// TIA Portal project "Stat Remp 2essay" (V15)

(* hardware
DEVICE "HMI_1"  TP1200 Comfort
   slot 0: "HMI_1"  TP1200 Comfort  6AV2 124-0MC01-0AX0  15.0.0.0
   slot 1: "HMI_RT_1"  TP1200 Comfort  6AV2 124-0MC01-0AX0  15.0.0.0
   slot 5: "HMI_1.IE_CP_1"  PROFINET Interface  15.0.0.0
      slot 1: "Interface PROFINET_1"  PROFINET Interface
         slot 1: "Port_1"  Port
         slot 2: "Port_2"  Port
   slot 7: "HMI_1.MPI/DP_CP_1"  MPI/DP Interface  15.0.0.0
DEVICE "Station S7-1200_1"  S7-1200 Station
   slot 0: "Châssis_0"  S7-1200 Rack  Rack  V1.0
   slot 1: "PLC_1"  CPU 1214C DC/DC/DC  6ES7 214-1AG40-0XB0  V4.2
*)

// ===== PLC "PLC_1"  CPU 1214C DC/DC/DC =====

VAR_GLOBAL   // PLC tag table "Table de variables standard"
   "System_Byte" AT %MB1 : Byte;
   "FirstScan" AT %M1.0 : Bool;
   "DiagStatusUpdate" AT %M1.1 : Bool;
   "AlwaysTRUE" AT %M1.2 : Bool;
   "AlwaysFALSE" AT %M1.3 : Bool;
   "Clock_Byte" AT %MB0 : Byte;
   "Clock_10Hz" AT %M0.0 : Bool;
   "Clock_5Hz" AT %M0.1 : Bool;
   "Clock_2.5Hz" AT %M0.2 : Bool;
   "Clock_2Hz" AT %M0.3 : Bool;
   "Clock_1.25Hz" AT %M0.4 : Bool;
   "Clock_1Hz" AT %M0.5 : Bool;
   "Clock_0.625Hz" AT %M0.6 : Bool;
   "Clock_0.5Hz" AT %M0.7 : Bool;
   "X1" AT %M2.0 : Bool;
   "V1" AT %Q0.0 : Bool;
   "X2" AT %M2.1 : Bool;
   "V3" AT %Q0.1 : Bool;
   "X3" AT %M2.2 : Bool;
   "V2" AT %Q0.2 : Bool;
   "MM" AT %Q0.3 : Bool;
   "X4" AT %M2.3 : Bool;
   "X5" AT %M2.4 : Bool;
   "MP" AT %Q0.4 : Bool;
   "X6" AT %M2.5 : Bool;
   "V6" AT %Q0.5 : Bool;
   "X7" AT %M2.6 : Bool;
   "MDR" AT %Q0.6 : Bool;
   "X8" AT %M2.7 : Bool;
   "DC" AT %Q0.7 : Bool;
   "X9" AT %M3.0 : Bool;
   "MG" AT %Q1.0 : Bool;
   "M-PT100" AT %MW4 : Int;
   "NICH" AT %MD6 : Real;
   "TMP" AT %MW10 : Int;
   "NIVEAU" AT %MW12 : Int;
   "NIV" AT %MD14 : Real;
   "M-NIVEAU" AT %MW18 : Int;
   "X0" AT %M3.1 : Bool;
   "forçage" AT %M3.2 : Bool;
   "L50" AT %M3.3 : Bool;
   "L400" AT %M3.4 : Bool;
   "L900" AT %M3.5 : Bool;
   "MA" AT %M3.6 : Bool;
   "MIN1" AT %M3.7 : Bool;
   "MAX1" AT %M20.0 : Bool;
   "FC-CHARG" AT %M20.1 : Bool;
   "MAXC" AT %M20.2 : Bool;
   "FC-DECH" AT %M20.3 : Bool;
   "VASC" AT %Q1.1 : Bool;
   "VADN" AT %Q1.2 : Bool;
   "THR-P" AT %M20.4 : Bool;
   "VAP" AT %Q1.3 : Bool;
   "ALARME" AT %M56.0 : Bool;
   "Acquitt-Btn" AT %M20.5 : Bool;
   "Acquittement" AT %M58.0 : Bool;
   "Res-Alr" AT %M20.6 : Bool;
   "Stop" AT %M20.7 : Bool;
   "Mot-Alarme" AT %MW56 : Int;
   "Mot-Acquittement" AT %MW58 : Int;
END_VAR

// folder: System blocks/Program resources

DATA_BLOCK "T1"   // DB1
{ S7_Optimized_Access := 'TRUE' }
AUTHOR : Simatic
FAMILY : IEC
NAME : IEC_TMR
VERSION : 1.0
// stored: InstanceOfName IEC_TIMER
"IEC_TIMER"
BEGIN
END_DATA_BLOCK

DATA_BLOCK "T2"   // DB2
{ S7_Optimized_Access := 'TRUE' }
AUTHOR : Simatic
FAMILY : IEC
NAME : IEC_TMR
VERSION : 1.0
// stored: InstanceOfName IEC_TIMER
"IEC_TIMER"
BEGIN
END_DATA_BLOCK

DATA_BLOCK "T3"   // DB3
{ S7_Optimized_Access := 'TRUE' }
AUTHOR : Simatic
FAMILY : IEC
NAME : IEC_TMR
VERSION : 1.0
// stored: InstanceOfName IEC_TIMER
"IEC_TIMER"
BEGIN
END_DATA_BLOCK

// folder: (top level)

FUNCTION "Actions" : Void   // FC1, LAD
{ S7_Optimized_Access := 'TRUE' }
VERSION : 0.1
   VAR_TEMP   // added for the SCL form of the ladder/FBD networks
      _w1 : Bool;
   END_VAR
BEGIN

REGION Network 1
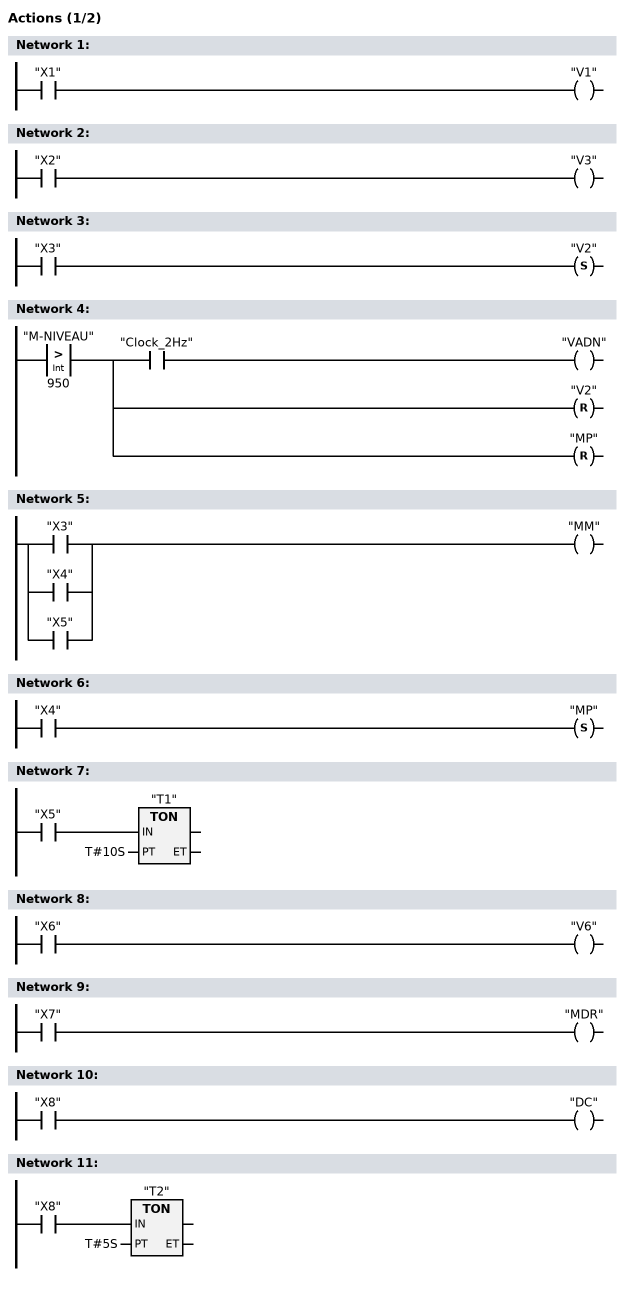
   RUNG wire#powerrail
      Contact( "X1" )
      Coil( "V1" )
   END_RUNG
   // the same network as SCL:
   "V1" := "X1";
END_REGION

REGION Network 2
   RUNG wire#powerrail
      Contact( "X2" )
      Coil( "V3" )
   END_RUNG
   // the same network as SCL:
   "V3" := "X2";
END_REGION

REGION Network 3
   RUNG wire#powerrail
      Contact( "X3" )
      S_Coil( "V2" )
   END_RUNG
   // the same network as SCL:
   IF "X3" THEN "V2" := TRUE; END_IF;
END_REGION

REGION Network 4
   RUNG wire#powerrail
      { S7_Templates := "SrcType := Int" } GT_Contact(in1 := "M-NIVEAU", in2 := 950)
      wire#w1
      Contact( "Clock_2Hz" )
      Coil( "VADN" )
   END_RUNG
   RUNG wire#w1
      R_Coil( "V2" )
   END_RUNG
   RUNG wire#w1
      R_Coil( "MP" )
   END_RUNG
   // the same network as SCL:
   #_w1 := "M-NIVEAU" > 950;
   "VADN" := #_w1 AND "Clock_2Hz";
   IF #_w1 THEN
       "V2" := FALSE;
       "MP" := FALSE;
   END_IF;
END_REGION

REGION Network 5
   RUNG wire#powerrail
      Contact( "X3" )
      wire#w1
      Coil( "MM" )
   END_RUNG
   RUNG wire#powerrail
      Contact( "X4" )
   END_RUNG wire#w1
   RUNG wire#powerrail
      Contact( "X5" )
   END_RUNG wire#w1
   // the same network as SCL:
   "MM" := "X3" OR "X4" OR "X5";
END_REGION

REGION Network 6
   RUNG wire#powerrail
      Contact( "X4" )
      S_Coil( "MP" )
   END_RUNG
   // the same network as SCL:
   IF "X4" THEN "MP" := TRUE; END_IF;
END_REGION

REGION Network 7
   "T1".TON(IN := "X5", PT := T#10S);
END_REGION

REGION Network 8
   RUNG wire#powerrail
      Contact( "X6" )
      Coil( "V6" )
   END_RUNG
   // the same network as SCL:
   "V6" := "X6";
END_REGION

REGION Network 9
   RUNG wire#powerrail
      Contact( "X7" )
      Coil( "MDR" )
   END_RUNG
   // the same network as SCL:
   "MDR" := "X7";
END_REGION

REGION Network 10
   RUNG wire#powerrail
      Contact( "X8" )
      Coil( "DC" )
   END_RUNG
   // the same network as SCL:
   "DC" := "X8";
END_REGION

REGION Network 11
   "T2".TON(IN := "X8", PT := T#5S);
END_REGION

REGION Network 12
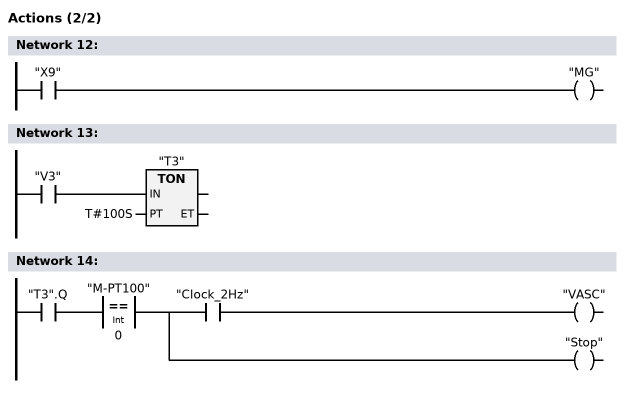
   RUNG wire#powerrail
      Contact( "X9" )
      Coil( "MG" )
   END_RUNG
   // the same network as SCL:
   "MG" := "X9";
END_REGION

REGION Network 13
   "T3".TON(IN := "V3", PT := T#100S);
END_REGION

REGION Network 14
   RUNG wire#powerrail
      Contact( "T3".Q )
      { S7_Templates := "SrcType := Int" } EQ_Contact(in1 := "M-PT100", in2 := 0)
      wire#w1
      Contact( "Clock_2Hz" )
      Coil( "VASC" )
   END_RUNG
   RUNG wire#w1
      Coil( "Stop" )
   END_RUNG
   // the same network as SCL:
   #_w1 := "T3".Q AND ("M-PT100" = 0);
   "VASC" := #_w1 AND "Clock_2Hz";
   "Stop" := #_w1;
END_REGION
END_FUNCTION

FUNCTION "Etapes" : Void   // FC2, LAD
{ S7_Optimized_Access := 'TRUE' }
VERSION : 0.1
BEGIN

REGION Network 1
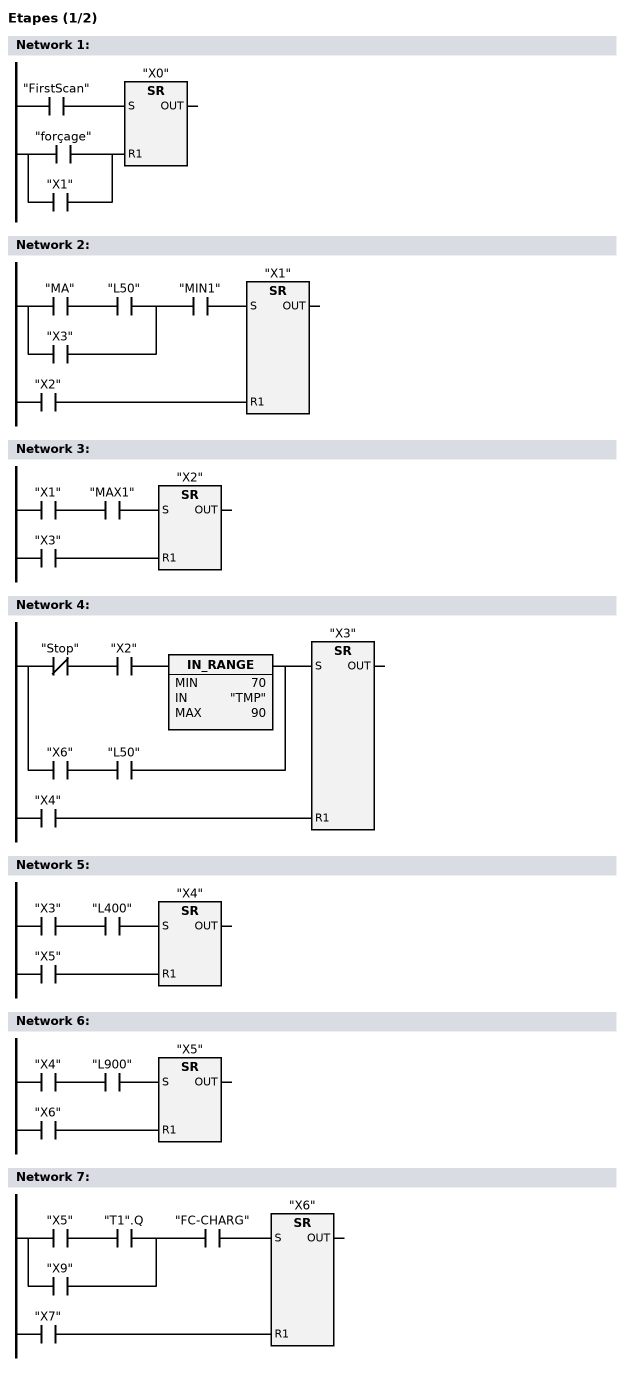
   RUNG wire#powerrail
      Contact( "FirstScan" )
      S_SR(operand := "X0", r1 := wire#w1)
   END_RUNG
   RUNG wire#powerrail
      Contact( "forçage" )
   END_RUNG wire#w1
   RUNG wire#powerrail
      Contact( "X1" )
   END_RUNG wire#w1
   // the same network as SCL:
   IF "FirstScan" THEN
       "X0" := TRUE;   // SR flip-flop
   END_IF;
   IF "forçage" OR "X1" THEN "X0" := FALSE; END_IF;
END_REGION

REGION Network 2
   RUNG wire#powerrail
      Contact( "MA" )
      Contact( "L50" )
      wire#w1
      Contact( "MIN1" )
      S_SR(operand := "X1", r1 := wire#w2)
   END_RUNG
   RUNG wire#powerrail
      Contact( "X3" )
   END_RUNG wire#w1
   RUNG wire#powerrail
      Contact( "X2" )
   END_RUNG wire#w2
   // the same network as SCL:
   IF (("MA" AND "L50") OR "X3") AND "MIN1" THEN
       "X1" := TRUE;   // SR flip-flop
   END_IF;
   IF "X2" THEN "X1" := FALSE; END_IF;
END_REGION

REGION Network 3
   RUNG wire#powerrail
      Contact( "X1" )
      Contact( "MAX1" )
      S_SR(operand := "X2", r1 := wire#w1)
   END_RUNG
   RUNG wire#powerrail
      Contact( "X3" )
   END_RUNG wire#w1
   // the same network as SCL:
   IF "X1" AND "MAX1" THEN
       "X2" := TRUE;   // SR flip-flop
   END_IF;
   IF "X3" THEN "X2" := FALSE; END_IF;
END_REGION

REGION Network 4
   RUNG wire#powerrail
      I_Contact( "Stop" )
      Contact( "X2" )
      { S7_Templates := "SrcType := Int" } InRange(min := 70, in := "TMP", max := 90)
      wire#w1
      S_SR(operand := "X3", r1 := wire#w2)
   END_RUNG
   RUNG wire#powerrail
      Contact( "X6" )
      Contact( "L50" )
   END_RUNG wire#w1
   RUNG wire#powerrail
      Contact( "X4" )
   END_RUNG wire#w2
   // the same network as SCL:
   IF (NOT "Stop" AND "X2" AND (70 <= "TMP") AND ("TMP" <= 90)) OR ("X6" AND "L50") THEN
       "X3" := TRUE;   // SR flip-flop
   END_IF;
   IF "X4" THEN "X3" := FALSE; END_IF;
END_REGION

REGION Network 5
   RUNG wire#powerrail
      Contact( "X3" )
      Contact( "L400" )
      S_SR(operand := "X4", r1 := wire#w1)
   END_RUNG
   RUNG wire#powerrail
      Contact( "X5" )
   END_RUNG wire#w1
   // the same network as SCL:
   IF "X3" AND "L400" THEN
       "X4" := TRUE;   // SR flip-flop
   END_IF;
   IF "X5" THEN "X4" := FALSE; END_IF;
END_REGION

REGION Network 6
   RUNG wire#powerrail
      Contact( "X4" )
      Contact( "L900" )
      S_SR(operand := "X5", r1 := wire#w1)
   END_RUNG
   RUNG wire#powerrail
      Contact( "X6" )
   END_RUNG wire#w1
   // the same network as SCL:
   IF "X4" AND "L900" THEN
       "X5" := TRUE;   // SR flip-flop
   END_IF;
   IF "X6" THEN "X5" := FALSE; END_IF;
END_REGION

REGION Network 7
   RUNG wire#powerrail
      Contact( "X5" )
      Contact( "T1".Q )
      wire#w1
      Contact( "FC-CHARG" )
      S_SR(operand := "X6", r1 := wire#w2)
   END_RUNG
   RUNG wire#powerrail
      Contact( "X9" )
   END_RUNG wire#w1
   RUNG wire#powerrail
      Contact( "X7" )
   END_RUNG wire#w2
   // the same network as SCL:
   IF (("X5" AND "T1".Q) OR "X9") AND "FC-CHARG" THEN
       "X6" := TRUE;   // SR flip-flop
   END_IF;
   IF "X7" THEN "X6" := FALSE; END_IF;
END_REGION

REGION Network 8
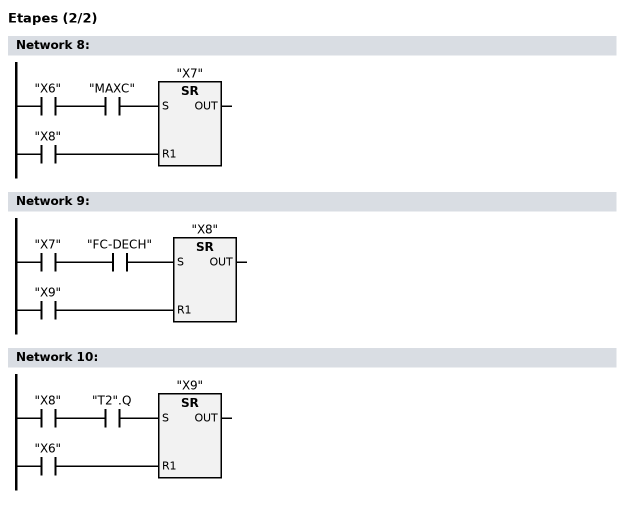
   RUNG wire#powerrail
      Contact( "X6" )
      Contact( "MAXC" )
      S_SR(operand := "X7", r1 := wire#w1)
   END_RUNG
   RUNG wire#powerrail
      Contact( "X8" )
   END_RUNG wire#w1
   // the same network as SCL:
   IF "X6" AND "MAXC" THEN
       "X7" := TRUE;   // SR flip-flop
   END_IF;
   IF "X8" THEN "X7" := FALSE; END_IF;
END_REGION

REGION Network 9
   RUNG wire#powerrail
      Contact( "X7" )
      Contact( "FC-DECH" )
      S_SR(operand := "X8", r1 := wire#w1)
   END_RUNG
   RUNG wire#powerrail
      Contact( "X9" )
   END_RUNG wire#w1
   // the same network as SCL:
   IF "X7" AND "FC-DECH" THEN
       "X8" := TRUE;   // SR flip-flop
   END_IF;
   IF "X9" THEN "X8" := FALSE; END_IF;
END_REGION

REGION Network 10
   RUNG wire#powerrail
      Contact( "X8" )
      Contact( "T2".Q )
      S_SR(operand := "X9", r1 := wire#w1)
   END_RUNG
   RUNG wire#powerrail
      Contact( "X6" )
   END_RUNG wire#w1
   // the same network as SCL:
   IF "X8" AND "T2".Q THEN
       "X9" := TRUE;   // SR flip-flop
   END_IF;
   IF "X6" THEN "X9" := FALSE; END_IF;
END_REGION
END_FUNCTION

FUNCTION "Traitement des grandeurs" : Void   // FC3, LAD
{ S7_Optimized_Access := 'TRUE' }
VERSION : 0.1
BEGIN

REGION Network 1
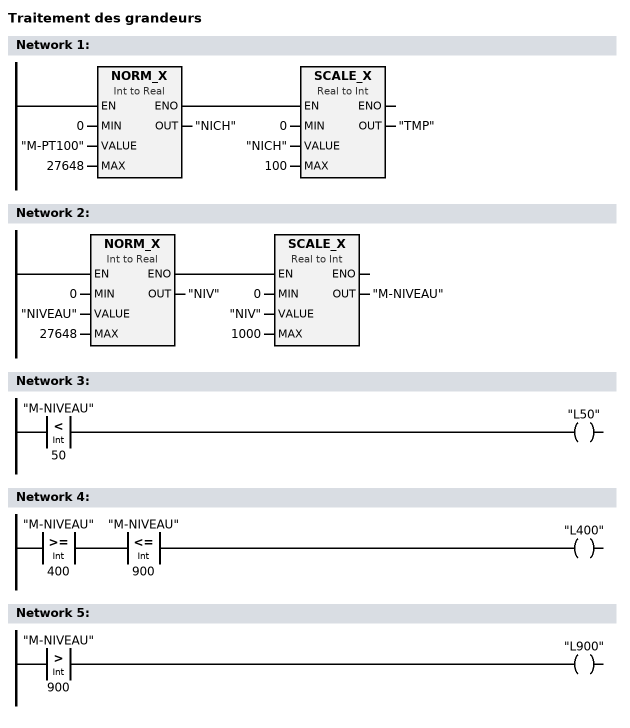
   RUNG wire#powerrail
      { S7_Templates := "[SrcType := Int, DestType := Real]" } Normalize(min := 0, value := "M-PT100", max := 27648, out => "NICH")
      { S7_Templates := "[SrcType := Real, DestType := Int]" } Scale(min := 0, value := "NICH", max := 100, out => "TMP")
   END_RUNG
   // the same network as SCL:
   "NICH" := NORM_X(MIN := 0, VALUE := "M-PT100", MAX := 27648);
   "TMP" := SCALE_X(MIN := 0, VALUE := "NICH", MAX := 100);
END_REGION

REGION Network 2
   RUNG wire#powerrail
      { S7_Templates := "[SrcType := Int, DestType := Real]" } Normalize(min := 0, value := "NIVEAU", max := 27648, out => "NIV")
      { S7_Templates := "[SrcType := Real, DestType := Int]" } Scale(min := 0, value := "NIV", max := 1000, out => "M-NIVEAU")
   END_RUNG
   // the same network as SCL:
   "NIV" := NORM_X(MIN := 0, VALUE := "NIVEAU", MAX := 27648);
   "M-NIVEAU" := SCALE_X(MIN := 0, VALUE := "NIV", MAX := 1000);
END_REGION

REGION Network 3
   RUNG wire#powerrail
      { S7_Templates := "SrcType := Int" } LT_Contact(in1 := "M-NIVEAU", in2 := 50)
      Coil( "L50" )
   END_RUNG
   // the same network as SCL:
   "L50" := "M-NIVEAU" < 50;
END_REGION

REGION Network 4
   RUNG wire#powerrail
      { S7_Templates := "SrcType := Int" } GE_Contact(in1 := "M-NIVEAU", in2 := 400)
      { S7_Templates := "SrcType := Int" } LE_Contact(in1 := "M-NIVEAU", in2 := 900)
      Coil( "L400" )
   END_RUNG
   // the same network as SCL:
   "L400" := ("M-NIVEAU" >= 400) AND ("M-NIVEAU" <= 900);
END_REGION

REGION Network 5
   RUNG wire#powerrail
      { S7_Templates := "SrcType := Int" } GT_Contact(in1 := "M-NIVEAU", in2 := 900)
      Coil( "L900" )
   END_RUNG
   // the same network as SCL:
   "L900" := "M-NIVEAU" > 900;
END_REGION
END_FUNCTION

FUNCTION "Alarmes" : Void   // FC4, LAD
{ S7_Optimized_Access := 'TRUE' }
VERSION : 0.1
BEGIN

REGION Network 1
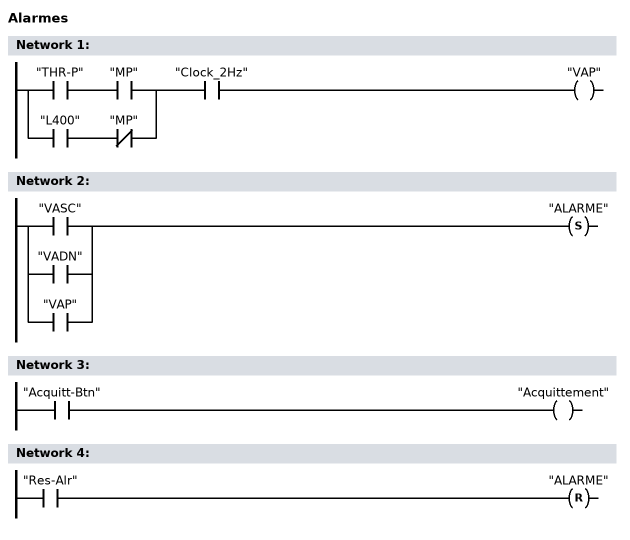
   RUNG wire#powerrail
      Contact( "THR-P" )
      Contact( "MP" )
      wire#w1
      Contact( "Clock_2Hz" )
      Coil( "VAP" )
   END_RUNG
   RUNG wire#powerrail
      Contact( "L400" )
      I_Contact( "MP" )
   END_RUNG wire#w1
   // the same network as SCL:
   "VAP" := (("THR-P" AND "MP") OR ("L400" AND NOT "MP")) AND "Clock_2Hz";
END_REGION

REGION Network 2
   RUNG wire#powerrail
      Contact( "VASC" )
      wire#w1
      S_Coil( "ALARME" )
   END_RUNG
   RUNG wire#powerrail
      Contact( "VADN" )
   END_RUNG wire#w1
   RUNG wire#powerrail
      Contact( "VAP" )
   END_RUNG wire#w1
   // the same network as SCL:
   IF "VASC" OR "VADN" OR "VAP" THEN "ALARME" := TRUE; END_IF;
END_REGION

REGION Network 3
   RUNG wire#powerrail
      Contact( "Acquitt-Btn" )
      Coil( "Acquittement" )
   END_RUNG
   // the same network as SCL:
   "Acquittement" := "Acquitt-Btn";
END_REGION

REGION Network 4
   RUNG wire#powerrail
      Contact( "Res-Alr" )
      R_Coil( "ALARME" )
   END_RUNG
   // the same network as SCL:
   IF "Res-Alr" THEN "ALARME" := FALSE; END_IF;
END_REGION
END_FUNCTION

ORGANIZATION_BLOCK "Main"   // OB1, LAD, ProgramCycle
TITLE = "Main Program Sweep (Cycle)"
{ S7_Optimized_Access := 'TRUE' }
VERSION : 0.1
   VAR_INPUT
      Initial_Call : Bool;   // Initial call of this OB
      Remanence : Bool;   // =True, if remanent data are available
   END_VAR
BEGIN

REGION Network 1
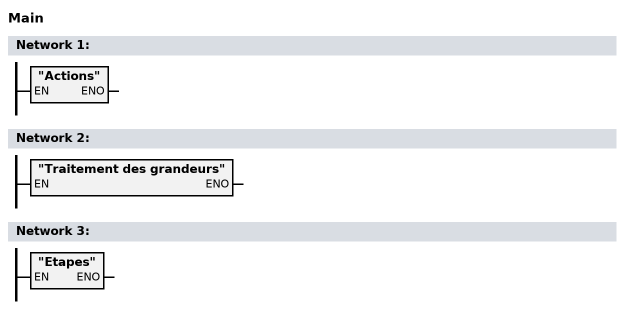
   RUNG wire#powerrail
      "Actions"()
   END_RUNG
   // the same network as SCL:
   "Actions"();
END_REGION

REGION Network 2
   RUNG wire#powerrail
      "Traitement des grandeurs"()
   END_RUNG
   // the same network as SCL:
   "Traitement des grandeurs"();
END_REGION

REGION Network 3
   RUNG wire#powerrail
      "Etapes"()
   END_RUNG
   // the same network as SCL:
   "Etapes"();
END_REGION
END_ORGANIZATION_BLOCK

(* ===== HMI "HMI_RT_1" =====
system functions are stored by id; their names below are inferred from use
connection "HMI_Liaison_1": ETHERNET, S7_1200_OMS

HMI tags "Table de variables standard"
   "Numéro_vue_variable" : UInt, internal
   "MP" : Bool = PLC MP AT %Q0.4, 1 s
   "V2" : Bool = PLC V2 AT %Q0.2, 1 s
   "Mot-Alarme" : Int = PLC "Mot-Alarme" AT %MW56, 1 s
   "Mot-Acquittement" : Int = PLC "Mot-Acquittement" AT %MW58, 1 s
   "MA" : Bool = PLC MA AT %M3.6, 1 s
   "forçage" : Bool = PLC forçage AT %M3.2, 1 s
   "M-PT100" : Int = PLC "M-PT100" AT %MW4, 1 s
   "TMP" : Int = PLC TMP AT %MW10, 1 s
   "NIVEAU" : Int = PLC NIVEAU AT %MW12, 1 s
   "M-NIVEAU" : Int = PLC "M-NIVEAU" AT %MW18, 1 s
   "V3" : Bool = PLC V3 AT %Q0.1, 1 s
   "V1" : Bool = PLC V1 AT %Q0.0, 1 s
   "MAX1" : Bool = PLC MAX1 AT %M20.0, 1 s
   "MIN1" : Bool = PLC MIN1 AT %M3.7, 1 s
   "MM" : Bool = PLC MM AT %Q0.3, 1 s
   "V6" : Bool = PLC V6 AT %Q0.5, 1 s
   "MAXC" : Bool = PLC MAXC AT %M20.2, 1 s
   "FC-CHARG" : Bool = PLC "FC-CHARG" AT %M20.1, 1 s
   "FC-DECH" : Bool = PLC "FC-DECH" AT %M20.3, 1 s
   "MDR" : Bool = PLC MDR AT %Q0.6, 1 s
   "MG" : Bool = PLC MG AT %Q1.0, 1 s
   "DC" : Bool = PLC DC AT %Q0.7, 1 s
   "VASC" : Bool = PLC VASC AT %Q1.1, 1 s
   "VADN" : Bool = PLC VADN AT %Q1.2, 1 s
   "VAP" : Bool = PLC VAP AT %Q1.3, 1 s
   "L50" : Bool = PLC L50 AT %M3.3, 1 s
   "L400" : Bool = PLC L400 AT %M3.4, 1 s
   "L900" : Bool = PLC L900 AT %M3.5, 1 s

discrete alarms
   1: 'Alarme detectée', class Errors, trigger "Mot-Alarme" bit 0

text list "Nom_vue_liste_textes": 1 'Vue racine'

screen "Vue racine" 1280x740, template "Modèle_1"
   on GenerateScreen: SetTag("Numéro_vue_variable", 1)
   Circle "Cercle_1" at 729,55 size 48x48
      Appearance <- "MP"
   Circle "Cercle_2" at 322,299 size 48x48
      Appearance <- "V2"
   Circle "Cercle_3" at 48,89 size 48x48
      Appearance <- "V1"
   TextField "Champ de texte_1" at 788,67 size 33x25; Text 'MP'
   TextField "Champ de texte_2" at 285,312 size 29x25; Text 'V2'
   Button "Bouton_1" at 1,573 size 192x32; TextOff 'Alarmes'
      on Click: ActivateScreen("Alarmes", 0)
   GraphicView "Vue de graphique_21" at 0,29 size 101x73; Picture "Graphique_3"
   GraphicView "Vue de graphique_22" at 97,19 size 65x67; Picture "Graphique_8"
   GraphicView "Vue de graphique_4" at 158,103 size 113x143; Picture "Graphique_5"
   GraphicView "Vue de graphique_11" at 465,316 size 184x90; Picture "Graphique_11"
   GraphicView "Vue de graphique_2" at 609,263 size 105x104; Picture "Graphique_2"
      Appearance <- "MM"
   GraphicView "Vue de graphique_3" at 698,106 size 76x77; Picture "Graphique_4"
   GraphicView "Vue de graphique_13" at 770,116 size 509x59; Picture "Graphique_3"
   GraphicView "Vue de graphique_23" at 197,27 size 49x79; Picture "Graphique_10"
   GraphicView "Vue de graphique_1" at 0,119 size 113x73; Picture "Graphique_3"
   GraphicView "Vue de graphique_5" at 98,107 size 65x69; Picture "Graphique_8"
   GraphicView "Vue de graphique_6" at 158,28 size 43x75; Picture "Graphique_3"
   Circle "Cercle_4" at 49,185 size 48x48
      Appearance <- "V3"
   GraphicView "Vue de graphique_8" at 190,242 size 49x75; Picture "Graphique_9"
   GraphicView "Vue de graphique_9" at 234,241 size 75x75; Picture "Graphique_3"
   GraphicView "Vue de graphique_10" at 306,232 size 65x67; Picture "Graphique_8"
   GraphicView "Vue de graphique_12" at 367,242 size 144x75; Picture "Graphique_3"
   GraphicView "Vue de graphique_14" at 510,240 size 49x79; Picture "Graphique_10"
   GraphicView "Vue de graphique_15" at 790,421 size 113x143; Picture "Graphique_5"
   GraphicView "Vue de graphique_16" at 563,95 size 43x53; Picture "Graphique_12"
   GraphicView "Vue de graphique_17" at 603,92 size 99x62; Picture "Graphique_3"
   GraphicView "Vue de graphique_18" at 563,145 size 45x176; Picture "Graphique_13"
   TextField "Champ de texte_3" at 678,337 size 37x25; Text 'MM'
   Circle "Cercle_5" at 710,312 size 48x48
      Appearance <- "MM"
   GraphicView "Vue de graphique_19" at 644,348 size 105x73; Picture "Graphique_3"
   GraphicView "Vue de graphique_20" at 745,337 size 65x67; Picture "Graphique_8"
   GraphicView "Vue de graphique_25" at 808,345 size 49x79; Picture "Graphique_10"
   TextField "Champ de texte_4" at 0,102 size 29x25; Text 'V1'
   TextField "Champ de texte_5" at 1,193 size 29x25; Text 'V3'
   Ellipse "Ellipse_1" at 268,101 size 53x28
      Appearance <- "MAX1"
   Ellipse "Ellipse_2" at 268,211 size 53x28
      Appearance <- "MIN1"
   Ellipse "Ellipse_3" at 937,565 size 53x28
      Appearance <- "FC-DECH"
   Ellipse "Ellipse_4" at 770,565 size 53x28
      Appearance <- "FC-CHARG"
   Ellipse "Ellipse_5" at 908,424 size 53x28
      Appearance <- "MAXC"
   Ellipse "Ellipse_6" at 768,605 size 53x28
      Appearance <- "MDR"
   Ellipse "Ellipse_7" at 937,605 size 53x28
      Appearance <- "MG"
   TextField "Champ de texte_6" at 682,563 size 88x25; Text 'FC-CHAR'
   TextField "Champ de texte_7" at 694,605 size 35x25; Text 'MD'
   TextField "Champ de texte_8" at 850,563 size 87x25; Text 'FC-DECH'
   TextField "Champ de texte_9" at 868,608 size 35x25; Text 'MG'
   TextField "Champ de texte_10" at 967,424 size 59x25; Text 'MAXC'
   TextField "Champ de texte_11" at 326,91 size 59x25; Text 'MAX1'
   TextField "Champ de texte_12" at 325,208 size 56x25; Text 'MIN1'
   Button "Bouton_2" at 1,335 size 96x32; TextOff 'MARCHE'
      on Press: SetBit("MA")
      on Release: ResetBit("MA")
   Button "Bouton_3" at 109,335 size 96x32; TextOff 'ARRET'
      on Click: SetBit("forçage")
   IOField "Champ d'E/S_1" at 10,425 size 96x32; FormatPattern s99999
      ProcessValue <- "M-PT100"
   IOField "Champ d'E/S_2" at 141,531 size 96x32; FormatPattern s99999
      ProcessValue <- "M-NIVEAU"
   IOField "Champ d'E/S_3" at 140,425 size 96x32; FormatPattern s99999
      ProcessValue <- "TMP"
   IOField "Champ d'E/S_4" at 8,531 size 96x32; FormatPattern s99999
      ProcessValue <- "NIVEAU"
   TextField "Champ de texte_13" at 24,393 size 72x25; Text 'PT-100'
   TextField "Champ de texte_14" at 162,395 size 44x25; Text 'TMP'
   TextField "Champ de texte_15" at 145,504 size 102x25; Text 'M-NIVEAU'
   TextField "Champ de texte_16" at 30,505 size 78x25; Text 'NIVEAU'
   Circle "Cercle_6" at 743,409 size 48x48
      Appearance <- "V6"
   TextField "Champ de texte_17" at 714,421 size 29x25; Text 'V6'
   TextField "Champ de texte_18" at 714,481 size 31x25; Text 'DC'
   Circle "Cercle_7" at 743,471 size 48x48
      Appearance <- "DC"
   Circle "Cercle_8" at 465,404 size 48x48
      Appearance <- "L50"
   Circle "Cercle_9" at 530,405 size 48x48
      Appearance <- "L400"
   Circle "Cercle_10" at 589,404 size 48x48
      Appearance <- "L900"
   TextField "Champ de texte_19" at 468,450 size 40x25; Text 'L50'
   TextField "Champ de texte_20" at 529,453 size 52x25; Text 'L400'
   TextField "Champ de texte_21" at 595,452 size 52x25; Text 'L900'

Template "Modèle_1" 1280x740
   Button "Quitter" at 1200,679 size 78x59; TextOff 'Quitter'; PictureOff "ExitRuntime_TP1200_Comfort_TR"; PictureOn "ExitRuntime_TP1200_Comfort_TR"
      on Release: StopRuntime(0)
   Button "Template_Button" at 1120,679 size 78x59; TextOff 'Text'
   Button "Template_Button_1" at 1040,679 size 78x59; TextOff 'Text'
   Button "Template_Button_2" at 960,679 size 78x59; TextOff 'Text'
   Button "Template_Button_3" at 880,679 size 78x59; TextOff 'Text'
   Button "Template_Button_4" at 800,679 size 78x59; TextOff 'Text'
   Button "Template_Button_5" at 720,679 size 78x59; TextOff 'Text'
   Button "Template_Button_6" at 640,679 size 78x59; TextOff 'Text'
   Button "Template_Button_7" at 561,679 size 78x59; TextOff 'Text'
   Button "Template_Button_8" at 481,679 size 78x59; TextOff 'Text'
   Button "Template_Button_9" at 401,679 size 78x59; TextOff 'Text'
   Button "Template_Button_10" at 321,679 size 78x59; TextOff 'Text'
   Button "Template_Button_11" at 241,679 size 78x59; TextOff 'Text'
   Button "Template_Button_12" at 161,679 size 78x59; TextOff 'Text'
   Button "Template_Button_13" at 81,679 size 78x59; TextOff 'Text'
   Button "Vue initiale" at 1,679 size 78x59; TextOff 'Vue initiale'; PictureOff "NavigateHome_TP1200_Comfort_TR"; PictureOn "NavigateHome_TP1200_Comfort_TR"
      on Release: ActivateScreen("Vue racine", 0)

screen "Alarmes" 1280x740
   Circle "Cercle_1" at 76,144 size 48x48
      Appearance <- "VASC"
   Circle "Cercle_2" at 76,241 size 48x48
      Appearance <- "VADN"
   Circle "Cercle_3" at 76,339 size 48x48
      Appearance <- "VAP"
   Button "Bouton_1" at 4,414 size 142x32; TextOff 'Vue racine'
      on Click: ActivateScreen("Vue racine", 0)
   AlarmView "Vue des alarmes_1" at 159,0 size 622x446
   TextField "Champ de texte_1" at 77,119 size 54x25; Text 'VASC'
   TextField "Champ de texte_2" at 77,208 size 58x25; Text 'VADN'
   TextField "Champ de texte_3" at 77,300 size 42x25; Text 'VAP'
*)